PROGRAM En_service
VAR	Fb_En_Service1:FB_En_Service;	B_Secu_Marche,	B_Securites,	Arret_auto,	Arret_Centrale_Niveau_Bas:BOOL;
	TON_K_En_Service_Hydraulique,	TON_ok_pour_rearm_1,	TON_ok_pour_rearm_2,	TON_K_Broches:TON;
	TON_Pressostat_Air, 	TON_Air_Ok,	TON_Marche_Ventilateur_centrale,	Ton_arret_Machine_Automatique:TON;
	TON_Acces_Machine_1,	TON_Acces_Machine_2: TON;
	TP_Reset,	TP_Rearm_Secu_1,	TP_Rearm_Secu_2,	TP_Arret_auto,	TP_Arret_Niveau_Bas:TP;		Ton_Validation_Variateur_Centrale: TON;
	RE_Machine_en_service: R_TRIG;
	TON_rearm: TON;
END_VAR
VAR // added by the converter: edge detectors and wires of the graphical bodies
    _w1 : BOOL;
END_VAR

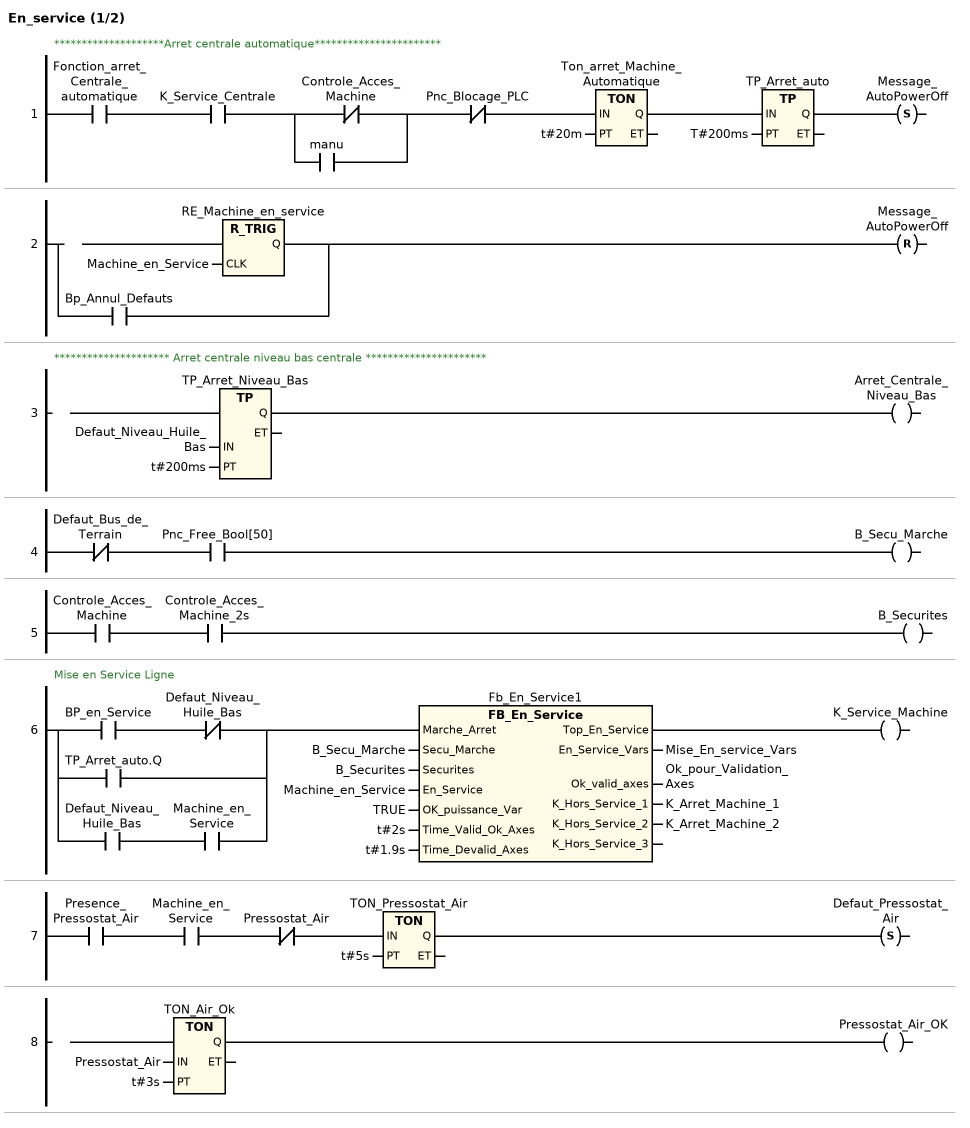
// NETWORK 1
// ********************Arret centrale automatique***********************
Ton_arret_Machine_Automatique(IN := (Fonction_arret_Centrale_automatique AND K_Service_Centrale AND (NOT Controle_Acces_Machine OR manu)) AND NOT Pnc_Blocage_PLC, PT := t#20m); // TON
TP_Arret_auto(IN := Ton_arret_Machine_Automatique.Q, PT := T#200ms); // TP
Message_AutoPowerOff S= TP_Arret_auto.Q;

// NETWORK 2
RE_Machine_en_service(CLK := Machine_en_Service); // R_TRIG
Message_AutoPowerOff R= RE_Machine_en_service.Q OR Bp_Annul_Defauts;

// NETWORK 3
// ********************* Arret centrale niveau bas centrale **********************
TP_Arret_Niveau_Bas(IN := Defaut_Niveau_Huile_Bas, PT := t#200ms); // TP
Arret_Centrale_Niveau_Bas := TP_Arret_Niveau_Bas.Q;

// NETWORK 4
B_Secu_Marche := NOT Defaut_Bus_de_Terrain AND Pnc_Free_Bool[50];

// NETWORK 5
B_Securites := Controle_Acces_Machine AND Controle_Acces_Machine_2s;

// NETWORK 6
// Mise en Service Ligne
Fb_En_Service1(
    Marche_Arret := BP_en_Service AND NOT Defaut_Niveau_Huile_Bas OR TP_Arret_auto.Q OR Defaut_Niveau_Huile_Bas AND Machine_en_Service,
    Secu_Marche := B_Secu_Marche,
    Securites := B_Securites,
    En_Service := Machine_en_Service,
    OK_puissance_Var := TRUE,
    Time_Valid_Ok_Axes := t#2s,
    Time_Devalid_Axes := t#1.9s,
    En_Service_Vars => Mise_En_service_Vars,
    Ok_valid_axes => Ok_pour_Validation_Axes,
    K_Hors_Service_1 => K_Arret_Machine_1,
    K_Hors_Service_2 => K_Arret_Machine_2); // FB_En_Service
K_Service_Machine := Fb_En_Service1.Top_En_Service;

// NETWORK 7
TON_Pressostat_Air(IN := Presence_Pressostat_Air AND Machine_en_Service AND NOT Pressostat_Air, PT := t#5s); // TON
Defaut_Pressostat_Air S= TON_Pressostat_Air.Q;

// NETWORK 8
TON_Air_Ok(IN := Pressostat_Air, PT := t#3s); // TON
Pressostat_Air_OK := TON_Air_Ok.Q;

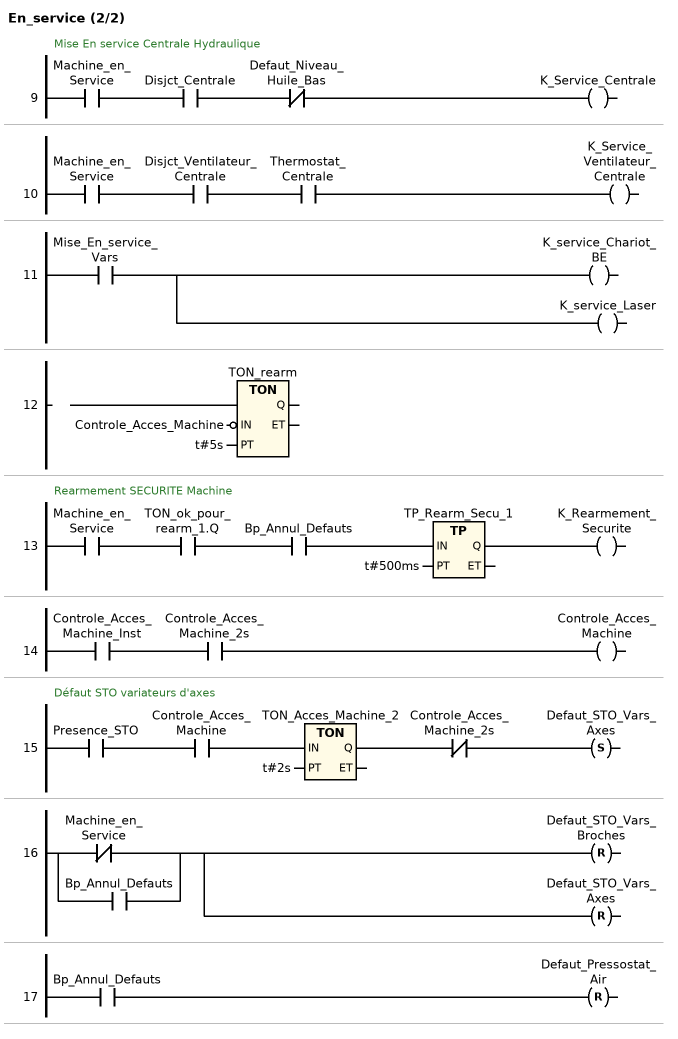
// NETWORK 9
// Mise En service Centrale Hydraulique
K_Service_Centrale := Machine_en_Service AND Disjct_Centrale AND NOT Defaut_Niveau_Huile_Bas;

// NETWORK 10
K_Service_Ventilateur_Centrale := Machine_en_Service AND Disjct_Ventilateur_Centrale AND Thermostat_Centrale;

// NETWORK 11
K_service_Chariot_BE := Mise_En_service_Vars;
K_service_Laser := Mise_En_service_Vars;

// NETWORK 12
TON_rearm(IN := NOT Controle_Acces_Machine, PT := t#5s); // TON

// NETWORK 13
// 					Rearmement SECURITE Machine
//
//
TP_Rearm_Secu_1(IN := Machine_en_Service AND TON_ok_pour_rearm_1.Q AND Bp_Annul_Defauts, PT := t#500ms); // TP
K_Rearmement_Securite := TP_Rearm_Secu_1.Q;

// NETWORK 14
Controle_Acces_Machine := Controle_Acces_Machine_Inst AND Controle_Acces_Machine_2s;

// NETWORK 15
// Défaut STO variateurs d'axes
TON_Acces_Machine_2(IN := Presence_STO AND Controle_Acces_Machine, PT := t#2s); // TON
Defaut_STO_Vars_Axes S= TON_Acces_Machine_2.Q AND NOT Controle_Acces_Machine_2s;

// NETWORK 16
_w1 := NOT Machine_en_Service OR Bp_Annul_Defauts;
Defaut_STO_Vars_Broches R= _w1;
Defaut_STO_Vars_Axes R= _w1;

// NETWORK 17
Defaut_Pressostat_Air R= Bp_Annul_Defauts;

END_PROGRAM

(* stored: Version 1.1.0.1
   POU En_service: Id {9816ed1a-dafd-4cfd-b0f2-e8afdefc0ff8}, SpecialFunc None *)
